// TIA Portal V19 export
TYPE "LEXCHANGETRAY_typePlasticEm5_toHandlingXyzRecieve"
// stored: Access Published
   STRUCT
      req { S7_SetPoint := 'True'} : "LEXCHANGETRAY_typeHandlingXyzEm_toPlasticReq";
   END_STRUCT;
END_TYPE
